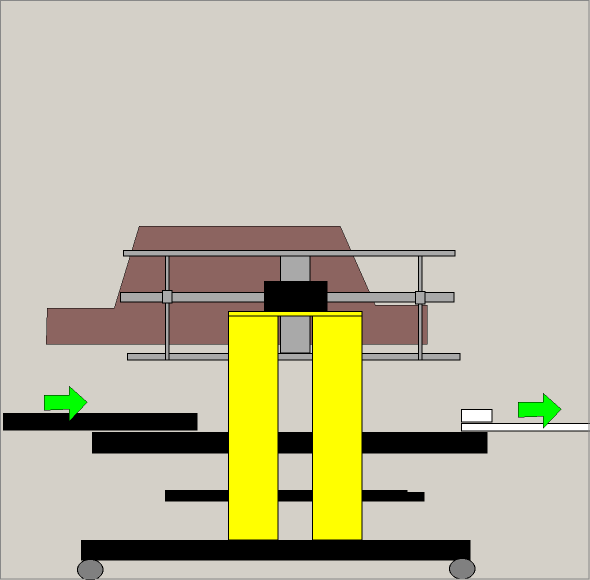
VISUALIZATION baseInSkiOutScreen  // 590x580
    Rectangle (461,423 130x8)
    Polygon (46,344) (47,308) (114,308) (139,226) (340,226) (375,305) (427,305) (427,343) (427,344)
    Rectangle (246,289 98x30), angle 90
    Rectangle (127,353 333x7)
    Rectangle (165,490 242x11), angle 25
    Rectangle (181,492 243x9), angle 336
    Rectangle (92,432 395x21)
    Rectangle (81,540 389x20)
    Rectangle (228,315 50x225)
    Rectangle (312,315 50x225)
    Ellipse (449,558 26x21)
    Ellipse (77,559 26x21)
    Rectangle (228,311 134x5)
    Rectangle (418,255 4x105)
    Rectangle (165,255 4x105)
    Rectangle (123,250 332x6)
    Rectangle (120,292 334x10)
    Rectangle (461,409 31x13)
    Rectangle (415,291 10x13)
    Rectangle (162,290 10x13)
    Rectangle (3,413 194x17)
    Polygon (44,405) (44,410) (69,409) (69,421) (87,402) (69,386) (69,395) (44,395)
    Polygon (518,412) (518,417) (543,416) (543,428) (561,409) (543,393) (543,402) (518,402)
    Rectangle (264,281 63x30)
END_VISUALIZATION

(* stored: Version 1.1.0.1, ProductVersion 3.1.4024.13
   Visu baseInSkiOutScreen: Id {a915e982-f28a-4c3a-80fa-7c1e24e1734f} *)
